FUNCTION_BLOCK ABSTRACT MatrixAccessor EXTENDS Matrix
VAR_INPUT
END_VAR
VAR_OUTPUT
END_VAR
VAR
	M_ : REFERENCE TO Matrix;
END_VAR

//Gets the value of the element in this matrix at the supplied location as if the elements were stored in a 1D row-major array
//:Prerequisites:
// - I < Rows*Cols
// - Matrix is not empty
//If the supplied index is out of bounds the value 0 is returned and a warning is generated in the Error List
METHOD PUBLIC GetI : LREAL//The value of the element at the specified index, or 0 if an invalid index is supplied
VAR_INPUT
	I : UINT;//The index of the element which should have its value returned
END_VAR
VAR
END_VAR
IF NOT __ISVALIDREF(M_) THEN
	GetI := 0.0;
	LogWarning('%s Attempted I access to uninitialized Matrix Accessor');
ELSIF IsEmpty THEN
	GetI := 0.0;
	LogWarning('%s: Attempted I access of empty Matrix Accessor');
ELSIF I >= Length THEN
	GetI := 0.0;
	LogWarning('%s: Attempted I access beyond limits of Matrix Accessor');
ELSE
	GetI := M_.GetI(This2Parent(I));
END_IF
END_METHOD

METHOD PROTECTED Init_
VAR_INPUT
	M : REFERENCE TO Matrix;
END_VAR
M_ REF= M;
END_METHOD

//Sets the element specified by the supplied index to the suppleid value, assuming the data of the matrix is stored in a 1D row-major array
//:Prerequisites: - I < Rows*Cols
METHOD PUBLIC SetI : BOOL//TRUE if the specified index is valid and the data is copied. FLASE otherwise
VAR_INPUT
	I : UINT;//The index specifying which element should be modified
	Val : LREAL;//The value copied to the corresponding element
END_VAR
IF NOT __ISVALIDREF(M_) THEN
	SetI := FALSE;
	LogWarning('%s Attempted I access to uninitialized Matrix Accessor');
ELSIF IsEmpty THEN
	SetI := FALSE;
	LogWarning('%s: Attempted I access of empty Matrix Accessor');
ELSIF I >= Length THEN
	SetI := FALSE;
	LogWarning('%s: Attempted I access beyond limits of Matrix Accessor');
ELSE
	SetI := M_.SetI(This2Parent(I),Val);
END_IF
END_METHOD

METHOD PROTECTED ABSTRACT This2Parent : UINT
VAR_INPUT
	Index : UINT;
END_VAR
END_METHOD

END_FUNCTION_BLOCK

(* stored: Version 1.1.0.1, ProductVersion 3.1.4024.9
   POU MatrixAccessor: Id {e50a508d-f480-0127-320a-803982deccd5}, SpecialFunc None
   Folder Initializers: Id {28431d55-f1be-0820-297a-111eb6985dc1}
   Folder Mapping: Id {8ff0265d-dfed-0d78-3f8a-9dc33a327da3}
   Folder Overrides: Id {8f59b246-ef31-06b6-3efd-d819bffceb36}
   Method GetI: Id {673a605f-ea3d-0fd4-108f-3cd0177f6697}
   Method Init_: Id {9d2c7dae-b3ad-036a-18e1-5c95ffea17d1}
   Method SetI: Id {2a187707-0985-02db-070b-3fa74894917a}
   Method This2Parent: Id {dfb72d27-38c6-0ee1-3757-2606a49a2af4} *)
